(* LS Electric XG5000 project: Coffee_make *)
(* PLC LSPLC *)

(* Comments on direct variables
%MX1	원두리필시작
%MX2	원두부족알림
%MX3	물리필시작
%MX4	물부족알림
%MX5	우유리필시작
%MX6	우유부족알림
%MX7	초코부족알림
%MX8	카페부족알림
%MX9	물부족팝업
%MX10	원두부족팝업
%MX11	우유부족팝업
%MX21	환기
*)

PROGRAM NewProgram (* task: 스캔 프로그램 *)
VAR
    on AT %IX0.0.0 : BOOL;
    timer : TON;
    timer10 : TON;
    timer11 : TON;
    timer12 : TON;
    timer13 : TON;
    timer14 : TON;
    timer17 : TP;
    timer17_1 : TON;
    timer18 : TP;
    timer18_1 : TON;
    timer19 : TP;
    timer19_1 : TON;
    timer2 : TON;
    timer3 : TON;
    timer4 : TON;
    timer5 : TON;
    timer6 : TON;
    timer7 : TON;
    timer8 : TON;
    timer9 : TON;
    tp : TP;
    tp1 : TP;
    tp2 : TP;
    tp3 : TP;
    tp4 : TP;
    가스경고 : BOOL;
    경찰신고 AT %MX81 : BOOL;
    공기정화 AT %MX22 : BOOL;
    근접센서1 AT %MX450 : BOOL;
    근접센서2 : BOOL;
    끊어줌 : BOOL;
    끊어줌_TOF : TOF;
    끓인물투입통과 : BOOL;
    나감 AT %IX0.0.24 : BOOL;
    다음으로 : BOOL;
    다음으로자가유지 : BOOL;
    대형1층동작 : TON;
    대형감지 AT %MX455 : BOOL;
    대형감지완료 AT %MX452 : BOOL;
    대형나감_TON : TON;
    대형도착 AT %QX0.1.27 : BOOL;
    대형엘리동작1 : TON;
    대형입장 AT %IX0.0.22 : BOOL;
    대형자동차나감 AT %QX0.1.45 : BOOL;
    대형자동차나감유지 : BOOL;
    대형자동차이동1 AT %QX0.1.43 : BOOL;
    대형자동차이동1_TON : TON;
    대형자동차이동2 AT %QX0.1.44 : BOOL;
    대형자동차이동2_TON : TON;
    대형키오스크_TON : TON;
    대형키오스크이동 AT %QX0.1.42 : BOOL;
    대형키오스크자기유지 : BOOL;
    도착 AT %QX0.1.31 : BOOL;
    뜨거운물투입TPQ AT %MX39 : BOOL;
    레일동작1 AT %QX0.1.47 : BOOL;
    레일동작1_TON : TON;
    레일동작2 AT %QX0.1.48 : BOOL;
    레일동작2_TON : TON;
    레일동작3 AT %QX0.1.49 : BOOL;
    레일동작3_TON : TON;
    레일동작4 AT %QX0.1.50 : BOOL;
    레일동작4_TON : TON;
    레일정지 AT %QX0.1.24 : BOOL;
    매장경고음 AT %MX80 : BOOL;
    멈춤 AT %IX0.0.26 : BOOL;
    물 AT %MW22 : INT;
    물끓이기 : TON;
    물끓이기TP : TP;
    물끓이기TPQ AT %MX38 : BOOL;
    물끓이기여부 AT %MX18 : BOOL;
    물무게 AT %MW11 : INT;
    물무게UDINT : UDINT;
    물무게곱하기 : INT;
    물투입 : TON;
    물투입1 : TON;
    물투입1TP : TP;
    물투입1TPQ AT %MX45 : BOOL;
    물투입TP : TP;
    물투입시간 : TIME;
    물투입여부 : BOOL;
    물투입통과 : BOOL;
    사이안화수소 : INT;
    섞기 : TON;
    섞기TP : TP;
    섞기TPQ AT %MX36 : BOOL;
    섞기통과 : BOOL;
    소형감지 AT %MX457 : BOOL;
    소형감지완료 AT %MX454 : BOOL;
    소형나감_TON : TON;
    소형도착 AT %QX0.1.25 : BOOL;
    소형입장 AT %IX0.0.20 : BOOL;
    소형자동차나감 AT %QX0.1.36 : BOOL;
    소형자동차나감유지 : BOOL;
    소형자동차이동1 AT %QX0.1.34 : BOOL;
    소형자동차이동2 AT %QX0.1.35 : BOOL;
    소형키오스크_TON : TON;
    소형키오스크이동 AT %QX0.1.33 : BOOL;
    소형키오스크자기유지 : BOOL;
    스프링쿨러 : BOOL;
    시럽무게곱하기 : INT;
    시럽용우유투입통과 : BOOL;
    시럽우유무게UDINT : UDINT;
    시럽우유투입 : TON;
    시럽우유투입TP : TP;
    시럽우유투입TPQ AT %MX37 : BOOL;
    시럽우유투입시간 : TIME;
    시작 : BOOL;
    실링기계 : TON;
    실링기계동작 : BOOL;
    실링레일 : TON;
    실링레일동작 AT %QX0.1.46 : BOOL;
    안끓인물투입통과 : BOOL;
    알림전송 AT %MX82 : BOOL;
    어딘가 : BOOL;
    얼음선투입 AT %MX16 : BOOL;
    얼음선투입TP : TP;
    얼음선투입TPQ AT %MX31 : BOOL;
    얼음선투입타이머 : TON;
    얼음선투입통과 : BOOL;
    얼음후투입 AT %MX17 : BOOL;
    얼음후투입TP : TP;
    얼음후투입TPQ AT %MX42 : BOOL;
    얼음후투입타이머 : TON;
    얼음후투입통과 : BOOL;
    에이드액무게 : INT := 0;
    에이드투입 : BOOL := 0;
    엘리1층도착 : BOOL;
    엘리내려감 AT %QX0.1.30 : BOOL;
    엘리베이터대기 : TON;
    엘리베이터동작 AT %QX0.1.28 : BOOL;
    엘리베이터중지 AT %QX0.1.29 : BOOL;
    연화수소 : INT;
    온도경고 : BOOL;
    온도센서 AT %MW83 : INT;
    우유 AT %MW24 : INT;
    우유뎁히기 : TON;
    우유뎁히기TP : TP;
    우유뎁히기TPQ AT %MX34 : BOOL;
    우유무게 AT %MW12 : INT := 0;
    우유무게UDINT : UDINT;
    우유무게곱하기 : INT;
    우유투입 : TON;
    우유투입1 : TON;
    우유투입2 : TON;
    우유투입2TP : TP;
    우유투입2TPQ AT %MX46 : BOOL;
    우유투입3 : TON;
    우유투입TP : TP;
    우유투입TPQ AT %MX35 : BOOL;
    우유투입시간 : TIME;
    우유투입시작 : BOOL;
    우유투입여부 : BOOL;
    우유투입통과 : BOOL;
    원두 AT %MW20 : INT;
    원두갈기 : TON;
    원두넣기 : TON;
    원두넣기시간 : TIME := T#5s;
    원두추출 : TON;
    유독가스해결 AT %MX52 : BOOL;
    유독경고 : BOOL;
    유독스위치 AT %MX55 : BOOL;
    유독안전 : BOOL;
    유독유지 : BOOL;
    유독주의 : BOOL;
    음료제조시작 AT %IX0.0.1 : BOOL;
    음료제조완료 AT %QX0.1.0 : BOOL;
    음료제조자가유지 : BOOL;
    이산화탄소 AT %MW84 : INT;
    이상감지 : BOOL;
    인체경고 : BOOL;
    일단멈춰 AT %QX0.1.51 : BOOL;
    일단멈춰2 : BOOL;
    일단멈춰3 : BOOL;
    일단멈춰4 : BOOL;
    일단멈춰5 : BOOL;
    일단멈춰6 : BOOL;
    일단멈춰7 : BOOL;
    일단멈춰8 : BOOL;
    일반우유투입통과 : BOOL;
    일산화탄소 : INT;
    자동차이동1_TON : TON;
    자동차이동2_TON : TON;
    자동차입장감지센서 AT %QX0.1.20 : BOOL;
    재고물 AT %MW23 : INT;
    재고우유 AT %MW25 : INT;
    재고원두 AT %MW21 : INT;
    재고초코 AT %MW26 : INT;
    재고카페 AT %MW27 : INT;
    전력 AT %MX20 : BOOL;
    전력스위치 AT %MX50 : BOOL;
    주차차단기개방 AT %QX0.1.21 : BOOL;
    주차차단기차단 AT %QX0.1.37 : BOOL;
    중형1층동작 : TON;
    중형감지 AT %MX456 : BOOL;
    중형감지완료 AT %MX453 : BOOL;
    중형나감_TON : TON;
    중형도착 AT %QX0.1.26 : BOOL;
    중형엘리동작1 : TON;
    중형입장 AT %IX0.0.21 : BOOL;
    중형자동차나감 AT %QX0.1.41 : BOOL;
    중형자동차나감유지 : BOOL;
    중형자동차이동1 AT %QX0.1.39 : BOOL;
    중형자동차이동1_TON : TON;
    중형자동차이동2 AT %QX0.1.40 : BOOL;
    중형자동차이동2_TON : TON;
    중형키오스크_TON : TON;
    중형키오스크이동 AT %QX0.1.38 : BOOL;
    중형키오스크자기유지 : BOOL;
    지나감감지 : TON;
    차량나감 AT %QX0.1.52 : BOOL;
    초기화 AT %IX0.0.25 : BOOL;
    초코시럽무게 AT %MW13 : INT;
    초코시럽무게UDINT : UDINT;
    초코시럽무게곱하기 : INT;
    초코시럽투입 : TON;
    초코시럽투입TP : TP;
    초코시럽투입TPQ AT %MX33 : BOOL;
    초코시럽투입시간 : TIME;
    초코시럽투입여부 : BOOL;
    초코시럽투입통과 : BOOL;
    카페시럽무게 AT %MW14 : INT := 0;
    카페시럽무게UDINT : UDINT;
    카페시럽무게곱하기 : INT;
    카페시럽투입 : TON;
    카페시럽투입1 : TON;
    카페시럽투입2 : TON;
    카페시럽투입TP : TP;
    카페시럽투입TPQ AT %MX32 : BOOL;
    카페시럽투입시간 : TIME;
    카페시럽투입여부 : BOOL;
    카페시럽투입통과 : BOOL;
    커피가레일로 : TON;
    커피가레일로2 : TON;
    커피가레일로2TP : TP;
    커피가레일로2TPQ AT %MX44 : BOOL;
    커피가레일로TP : TP;
    커피가레일로TPQ AT %MX43 : BOOL;
    커피끓이기시간 : TIME;
    커피무게 AT %MW10 : INT;
    커피무게UDINT : UDINT;
    커피무게곱하기 : INT;
    커피배달중 AT %QX0.1.32 : BOOL;
    커피온도 AT %MW15 : INT;
    커피온도UDINT : UDINT;
    커피온도곱하기 : INT;
    커피제작시작 AT %QX0.1.22 : BOOL;
    커피제작완료 AT %QX0.1.23 : BOOL;
    커피주문완료 AT %MX451 : BOOL;
    커피추출 : TON;
    커피추출TP : TP;
    커피추출TPQ AT %MX40 : BOOL;
    커피투입 : TON;
    커피투입TP : TP;
    커피투입TPQ AT %MX41 : BOOL;
    커피투입시간 : TIME;
    커피투입시작 : BOOL;
    커피투입통과 : BOOL;
    컵구멍인지 : TON;
    컵투입 : TON;
    컵투입TP : TP;
    컵투입TPQ AT %MX30 : BOOL;
    컵투입통과 AT %MX65 : BOOL;
    컵투하직후TP : TP;
    쿨러온 AT %MX53 : BOOL;
    타이머 : TON;
    타이머1 : TON;
    타이머2 : TON;
    타이머3 : TON;
    호퍼닫기 : BOOL;
    화재위험 : BOOL;
    화재진압 : BOOL;
    환기스위치 AT %MX51 : BOOL;
END_VAR
VAR
    _t1 : BOOL;
    _t2 : BOOL;
    _t3 : BOOL;
    _t4 : BOOL;
    _p5 : BOOL;
    _t6 : BOOL;
    _t7 : BOOL;
    _t8 : BOOL;
    _t9 : BOOL;
    _t10 : BOOL;
    _t11 : BOOL;
    _t12 : BOOL;
    _t13 : BOOL;
    _t14 : BOOL;
    _t15 : BOOL;
    _t16 : BOOL;
    _t17 : BOOL;
END_VAR

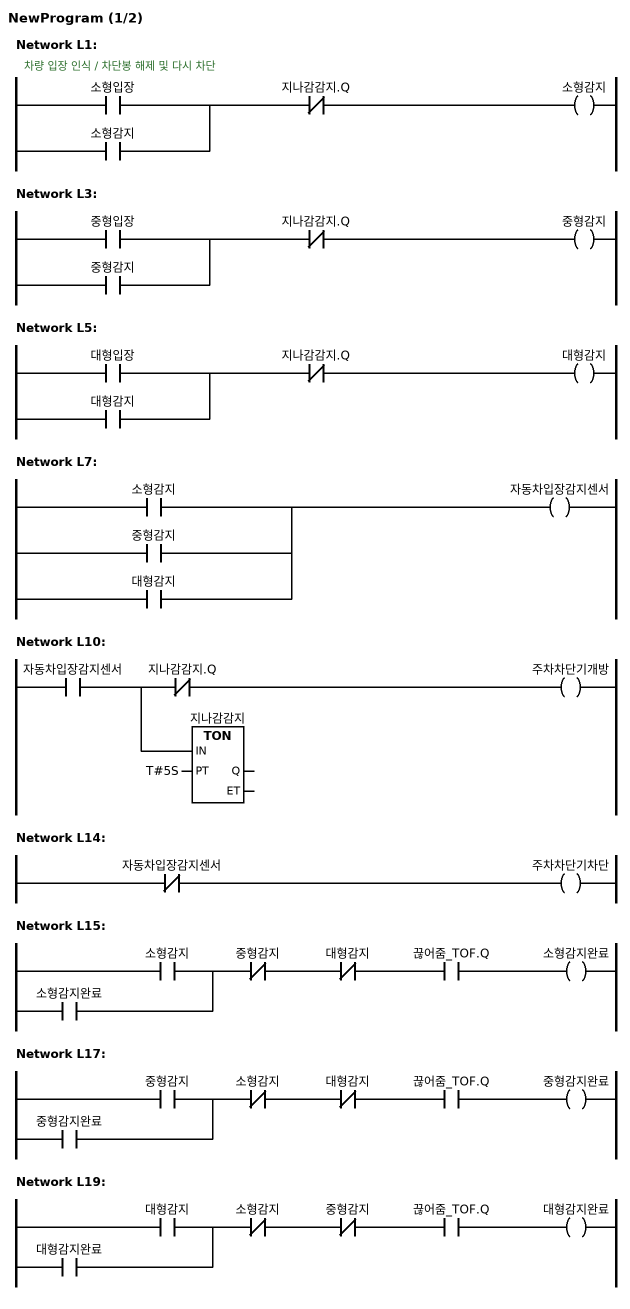
(* 차량 입장 인식 / 차단봉 해제 및 다시 차단 *)
(* Rung L1 *)
소형감지 := (소형입장 OR 소형감지) AND NOT 지나감감지.Q;
(* Rung L3 *)
중형감지 := (중형입장 OR 중형감지) AND NOT 지나감감지.Q;
(* Rung L5 *)
대형감지 := (대형입장 OR 대형감지) AND NOT 지나감감지.Q;
(* Rung L7 *)
자동차입장감지센서 := 소형감지 OR 중형감지 OR 대형감지;
(* Rung L10 *)
주차차단기개방 := 자동차입장감지센서 AND NOT 지나감감지.Q;
지나감감지(IN := 자동차입장감지센서, PT := T#5S);
(* Rung L14 *)
주차차단기차단 := NOT 자동차입장감지센서;
(* Rung L15 *)
소형감지완료 := (소형감지 OR 소형감지완료) AND NOT 중형감지 AND NOT 대형감지 AND 끊어줌_TOF.Q;
(* Rung L17 *)
중형감지완료 := (중형감지 OR 중형감지완료) AND NOT 소형감지 AND NOT 대형감지 AND 끊어줌_TOF.Q;
(* Rung L19 *)
대형감지완료 := (대형감지 OR 대형감지완료) AND NOT 소형감지 AND NOT 중형감지 AND 끊어줌_TOF.Q;

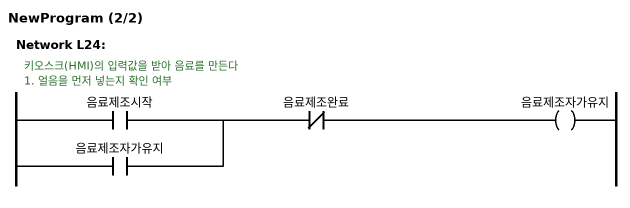
(* 키오스크(HMI)의 입력값을 받아 음료를 만든다 *)
(* 1. 얼음을 먼저 넣는지 확인 여부 *)
(* Rung L24 *)
음료제조자가유지 := (음료제조시작 OR 음료제조자가유지) AND NOT 음료제조완료;

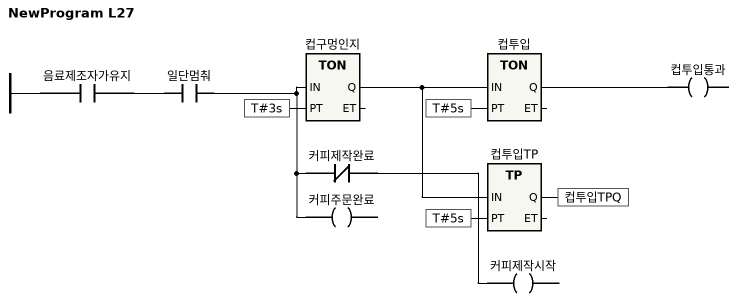
(* Rung L27 *)
커피제작시작 := 음료제조자가유지 AND 일단멈춰 AND NOT 커피제작완료;
커피주문완료 := 음료제조자가유지 AND 일단멈춰;
컵구멍인지(IN := 음료제조자가유지 AND 일단멈춰, PT := T#3s);
컵투입(IN := 컵구멍인지.Q, PT := T#5s);
컵투입통과 := 컵투입.Q;
컵투입TP(IN := 컵구멍인지.Q, PT := T#5s);
컵투입TPQ := 컵투입TP.Q;

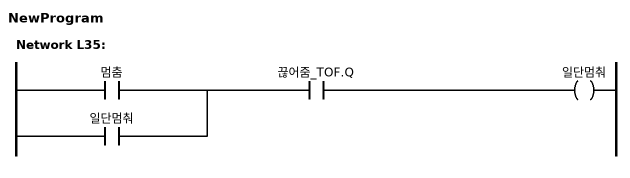
(* Rung L35 *)
일단멈춰 := (멈춤 OR 일단멈춰) AND 끊어줌_TOF.Q;

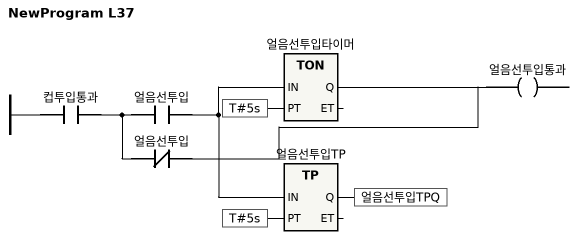
(* Rung L37 *)
얼음선투입타이머(IN := 컵투입통과 AND 얼음선투입, PT := T#5s);
얼음선투입통과 := 얼음선투입타이머.Q OR (컵투입통과 AND NOT 얼음선투입);
얼음선투입TP(IN := 컵투입통과 AND 얼음선투입, PT := T#5s);
얼음선투입TPQ := 얼음선투입TP.Q;

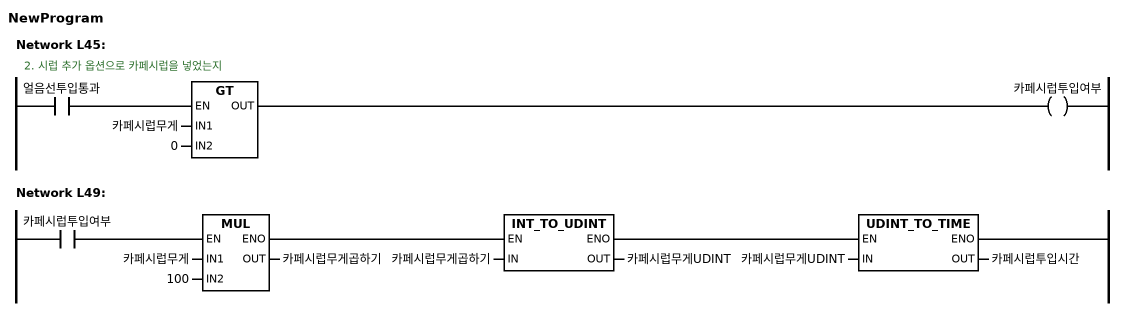
(* 2. 시럽 추가 옵션으로 카페시럽을 넣었는지 *)
(* Rung L45 *)
IF 얼음선투입통과 THEN _t1 := 카페시럽무게 > 0; END_IF;
카페시럽투입여부 := _t1;
(* Rung L49 *)
IF 카페시럽투입여부 THEN
    카페시럽무게곱하기 := 카페시럽무게 * 100;
    카페시럽무게UDINT := INT_TO_UDINT(카페시럽무게곱하기);
    카페시럽투입시간 := UDINT_TO_TIME(카페시럽무게UDINT);
END_IF;

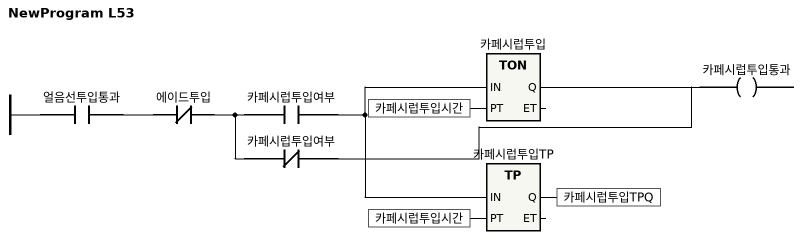
(* Rung L53 *)
카페시럽투입(IN := 얼음선투입통과 AND NOT 에이드투입 AND 카페시럽투입여부, PT := 카페시럽투입시간);
카페시럽투입통과 := 카페시럽투입.Q OR (얼음선투입통과 AND NOT 에이드투입 AND NOT 카페시럽투입여부);
카페시럽투입TP(IN := 얼음선투입통과 AND NOT 에이드투입 AND 카페시럽투입여부, PT := 카페시럽투입시간);
카페시럽투입TPQ := 카페시럽투입TP.Q;

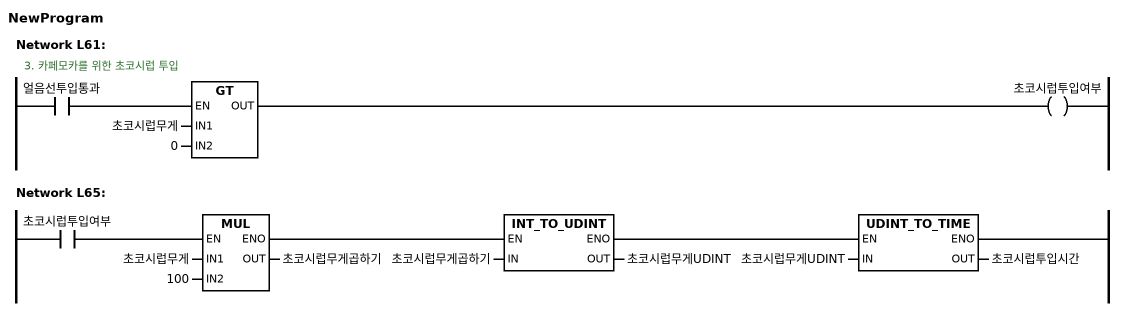
(* 3. 카페모카를 위한 초코시럽 투입 *)
(* Rung L61 *)
IF 얼음선투입통과 THEN _t2 := 초코시럽무게 > 0; END_IF;
초코시럽투입여부 := _t2;
(* Rung L65 *)
IF 초코시럽투입여부 THEN
    초코시럽무게곱하기 := 초코시럽무게 * 100;
    초코시럽무게UDINT := INT_TO_UDINT(초코시럽무게곱하기);
    초코시럽투입시간 := UDINT_TO_TIME(초코시럽무게UDINT);
END_IF;

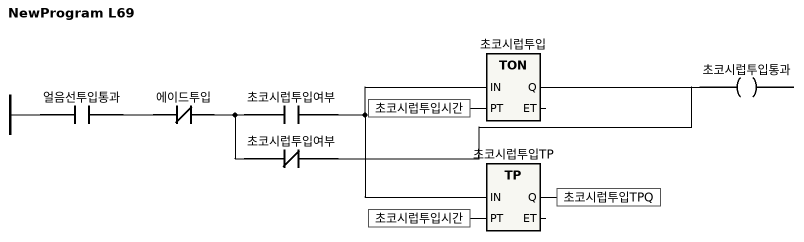
(* Rung L69 *)
초코시럽투입(IN := 얼음선투입통과 AND NOT 에이드투입 AND 초코시럽투입여부, PT := 초코시럽투입시간);
초코시럽투입통과 := 초코시럽투입.Q OR (얼음선투입통과 AND NOT 에이드투입 AND NOT 초코시럽투입여부);
초코시럽투입TP(IN := 얼음선투입통과 AND NOT 에이드투입 AND 초코시럽투입여부, PT := 초코시럽투입시간);
초코시럽투입TPQ := 초코시럽투입TP.Q;

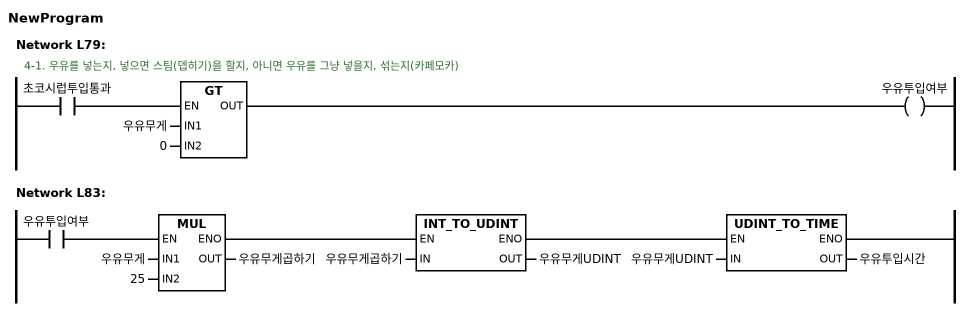
(* 4-1. 우유를 넣는지, 넣으면 스팀(뎁히기)을 할지, 아니면 우유를 그냥 넣을지, 섞는지(카페모카) *)
(* Rung L79 *)
IF 초코시럽투입통과 THEN _t3 := 우유무게 > 0; END_IF;
우유투입여부 := _t3;
(* Rung L83 *)
IF 우유투입여부 THEN
    우유무게곱하기 := 우유무게 * 25;
    우유무게UDINT := INT_TO_UDINT(우유무게곱하기);
    우유투입시간 := UDINT_TO_TIME(우유무게UDINT);
END_IF;

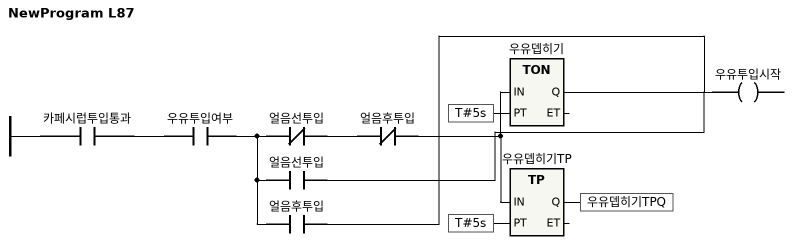
(* Rung L87 *)
우유뎁히기(IN := 카페시럽투입통과 AND 우유투입여부 AND NOT 얼음선투입 AND NOT 얼음후투입, PT := T#5s);
우유투입시작 := 우유뎁히기.Q OR (카페시럽투입통과 AND 우유투입여부 AND (얼음선투입 OR 얼음후투입));
우유뎁히기TP(IN := 카페시럽투입통과 AND 우유투입여부 AND NOT 얼음선투입 AND NOT 얼음후투입, PT := T#5s);
우유뎁히기TPQ := 우유뎁히기TP.Q;

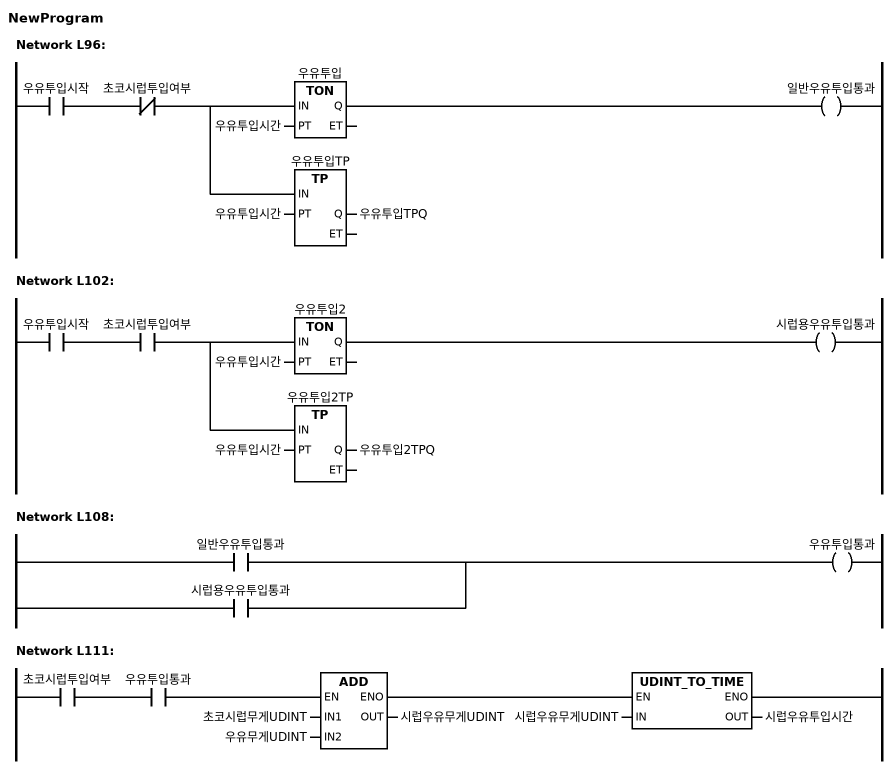
(* Rung L96 *)
우유투입(IN := 우유투입시작 AND NOT 초코시럽투입여부, PT := 우유투입시간);
일반우유투입통과 := 우유투입.Q;
우유투입TP(IN := 우유투입시작 AND NOT 초코시럽투입여부, PT := 우유투입시간, Q => 우유투입TPQ);
(* Rung L102 *)
우유투입2(IN := 우유투입시작 AND 초코시럽투입여부, PT := 우유투입시간);
시럽용우유투입통과 := 우유투입2.Q;
우유투입2TP(IN := 우유투입시작 AND 초코시럽투입여부, PT := 우유투입시간, Q => 우유투입2TPQ);
(* Rung L108 *)
우유투입통과 := 일반우유투입통과 OR 시럽용우유투입통과;
(* Rung L111 *)
IF 초코시럽투입여부 AND 우유투입통과 THEN
    시럽우유무게UDINT := 초코시럽무게UDINT + 우유무게UDINT;
    시럽우유투입시간 := UDINT_TO_TIME(시럽우유무게UDINT);
END_IF;

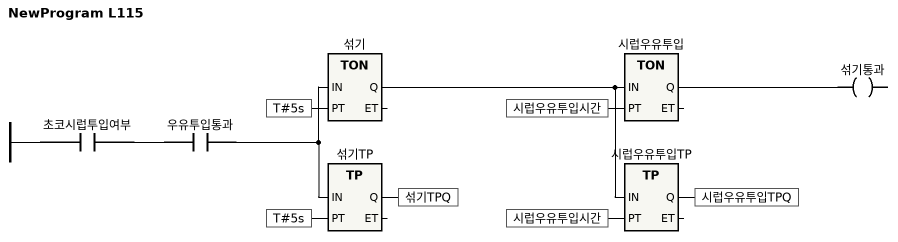
(* Rung L115 *)
섞기(IN := 초코시럽투입여부 AND 우유투입통과, PT := T#5s);
시럽우유투입(IN := 섞기.Q, PT := 시럽우유투입시간);
섞기통과 := 시럽우유투입.Q;
섞기TP(IN := 초코시럽투입여부 AND 우유투입통과, PT := T#5s);
섞기TPQ := 섞기TP.Q;
시럽우유투입TP(IN := 섞기.Q, PT := 시럽우유투입시간);
시럽우유투입TPQ := 시럽우유투입TP.Q;

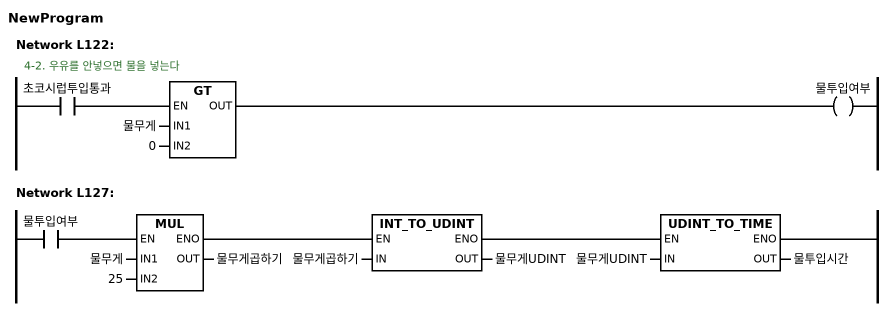
(* 4-2. 우유를 안넣으면 물을 넣는다 *)
(* Rung L122 *)
IF 초코시럽투입통과 THEN _t4 := 물무게 > 0; END_IF;
물투입여부 := _t4;
(* Rung L127 *)
IF 물투입여부 THEN
    물무게곱하기 := 물무게 * 25;
    물무게UDINT := INT_TO_UDINT(물무게곱하기);
    물투입시간 := UDINT_TO_TIME(물무게UDINT);
END_IF;

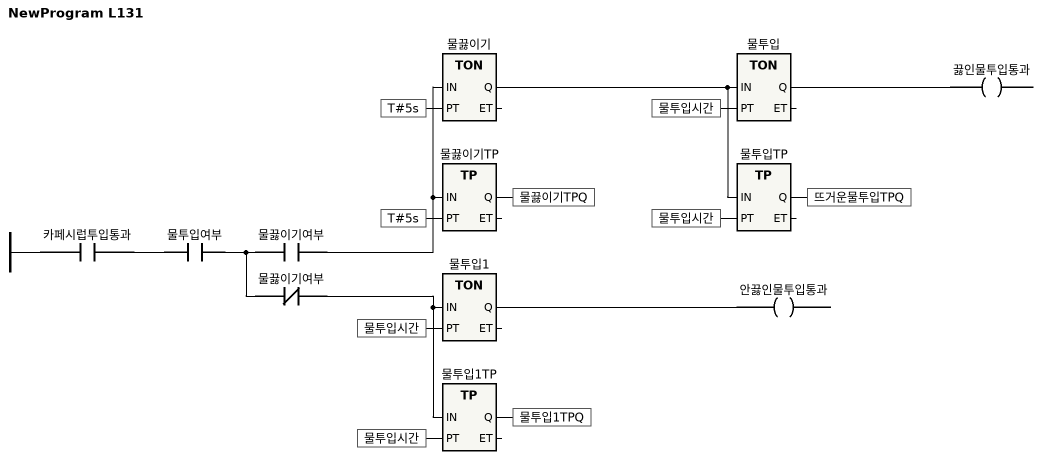
(* Rung L131 *)
물끓이기(IN := 카페시럽투입통과 AND 물투입여부 AND 물끓이기여부, PT := T#5s);
물투입(IN := 물끓이기.Q, PT := 물투입시간);
끓인물투입통과 := 물투입.Q;
물끓이기TP(IN := 카페시럽투입통과 AND 물투입여부 AND 물끓이기여부, PT := T#5s);
물끓이기TPQ := 물끓이기TP.Q;
물투입TP(IN := 물끓이기.Q, PT := 물투입시간);
뜨거운물투입TPQ := 물투입TP.Q;
물투입1(IN := 카페시럽투입통과 AND 물투입여부 AND NOT 물끓이기여부, PT := 물투입시간);
안끓인물투입통과 := 물투입1.Q;
물투입1TP(IN := 카페시럽투입통과 AND 물투입여부 AND NOT 물끓이기여부, PT := 물투입시간);
물투입1TPQ := 물투입1TP.Q;

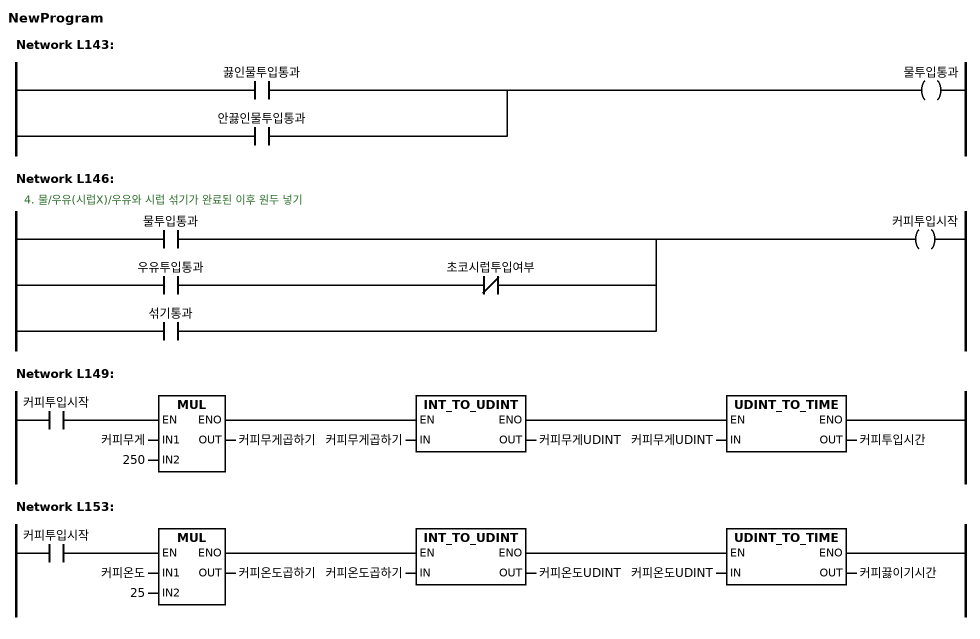
(* Rung L143 *)
물투입통과 := 끓인물투입통과 OR 안끓인물투입통과;
(* 4. 물/우유(시럽X)/우유와 시럽 섞기가 완료된 이후 원두 넣기 *)
(* Rung L146 *)
커피투입시작 := 물투입통과 OR (우유투입통과 AND NOT 초코시럽투입여부) OR 섞기통과;
(* Rung L149 *)
IF 커피투입시작 THEN
    커피무게곱하기 := 커피무게 * 250;
    커피무게UDINT := INT_TO_UDINT(커피무게곱하기);
    커피투입시간 := UDINT_TO_TIME(커피무게UDINT);
END_IF;
(* Rung L153 *)
IF 커피투입시작 THEN
    커피온도곱하기 := 커피온도 * 25;
    커피온도UDINT := INT_TO_UDINT(커피온도곱하기);
    커피끓이기시간 := UDINT_TO_TIME(커피온도UDINT);
END_IF;

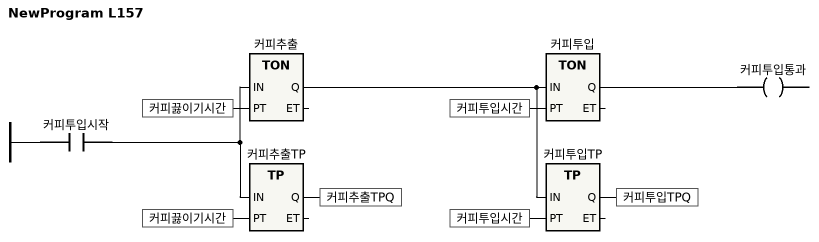
(* Rung L157 *)
커피추출(IN := 커피투입시작, PT := 커피끓이기시간);
커피투입(IN := 커피추출.Q, PT := 커피투입시간);
커피투입통과 := 커피투입.Q;
커피추출TP(IN := 커피투입시작, PT := 커피끓이기시간);
커피추출TPQ := 커피추출TP.Q;
커피투입TP(IN := 커피추출.Q, PT := 커피투입시간);
커피투입TPQ := 커피투입TP.Q;

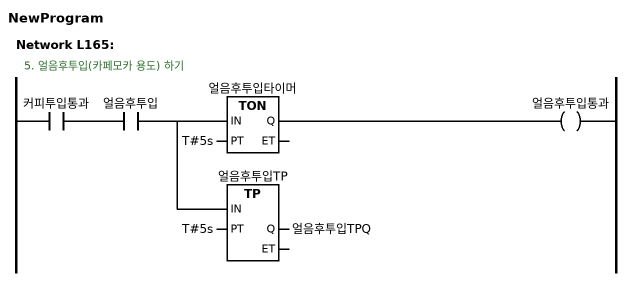
(* 5. 얼음후투입(카페모카 용도) 하기 *)
(* Rung L165 *)
얼음후투입타이머(IN := 커피투입통과 AND 얼음후투입, PT := T#5s);
얼음후투입통과 := 얼음후투입타이머.Q;
얼음후투입TP(IN := 커피투입통과 AND 얼음후투입, PT := T#5s, Q => 얼음후투입TPQ);

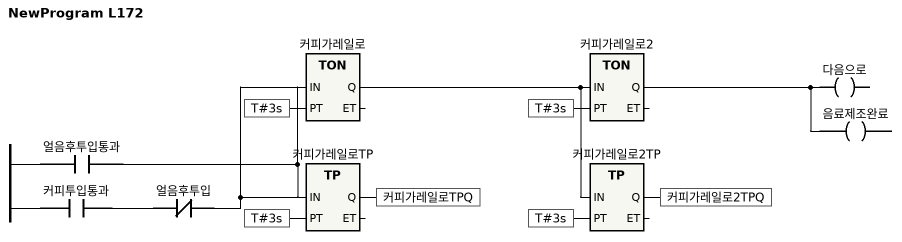
(* 끝. 음료제조완료 확인하기 *)
(* Rung L172 *)
커피가레일로(IN := 얼음후투입통과 OR (커피투입통과 AND NOT 얼음후투입), PT := T#3s);
커피가레일로2(IN := 커피가레일로.Q, PT := T#3s);
다음으로 := 커피가레일로2.Q;
음료제조완료 := 커피가레일로2.Q;
커피가레일로TP(IN := 얼음후투입통과 OR (커피투입통과 AND NOT 얼음후투입), PT := T#3s);
커피가레일로TPQ := 커피가레일로TP.Q;
커피가레일로2TP(IN := 커피가레일로.Q, PT := T#3s);
커피가레일로2TPQ := 커피가레일로2TP.Q;

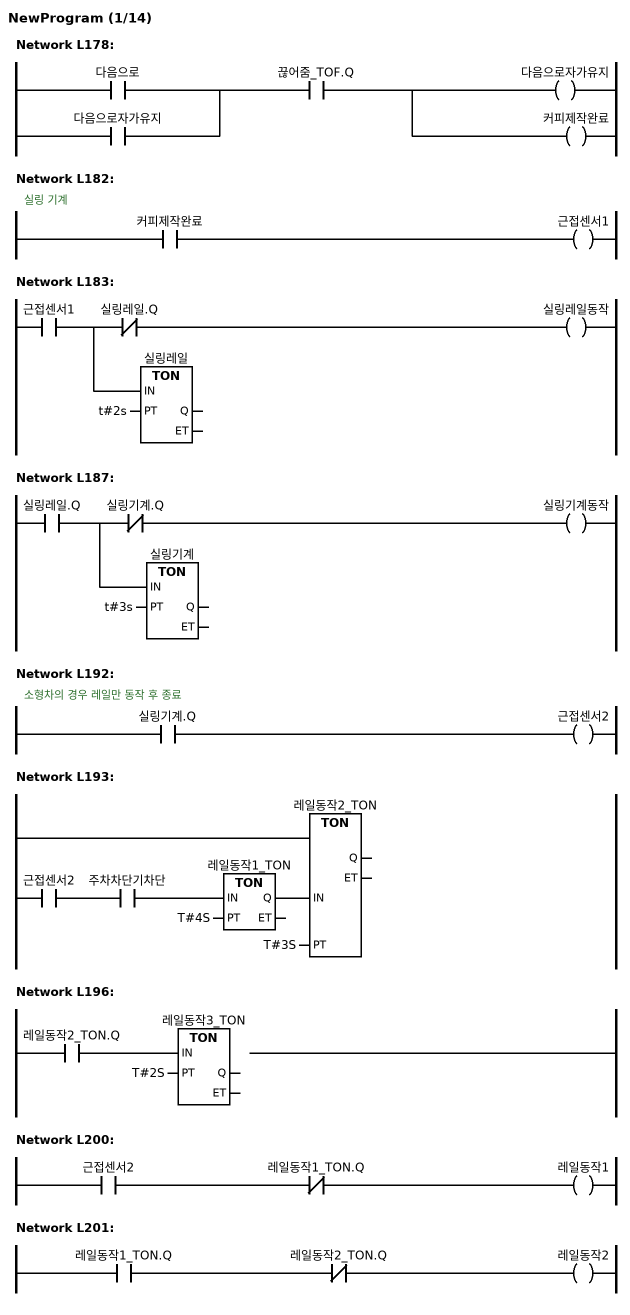
(* Rung L178 *)
_p5 := (다음으로 OR 다음으로자가유지) AND 끊어줌_TOF.Q;
다음으로자가유지 := _p5;
커피제작완료 := _p5;
(* 실링 기계 *)
(* Rung L182 *)
근접센서1 := 커피제작완료;
(* Rung L183 *)
실링레일동작 := 근접센서1 AND NOT 실링레일.Q;
실링레일(IN := 근접센서1, PT := t#2s);
(* Rung L187 *)
실링기계동작 := 실링레일.Q AND NOT 실링기계.Q;
실링기계(IN := 실링레일.Q, PT := t#3s);
(* 소형차의 경우 레일만 동작 후 종료 *)
(* Rung L192 *)
근접센서2 := 실링기계.Q;
(* Rung L193 *)
레일동작1_TON(IN := 근접센서2 AND 주차차단기차단, PT := T#4S);
레일동작2_TON(IN := 레일동작1_TON.Q, PT := T#3S);
(* Rung L196 *)
레일동작3_TON(IN := 레일동작2_TON.Q, PT := T#2S);
(* Rung L200 *)
레일동작1 := 근접센서2 AND NOT 레일동작1_TON.Q;
(* Rung L201 *)
레일동작2 := 레일동작1_TON.Q AND NOT 레일동작2_TON.Q;

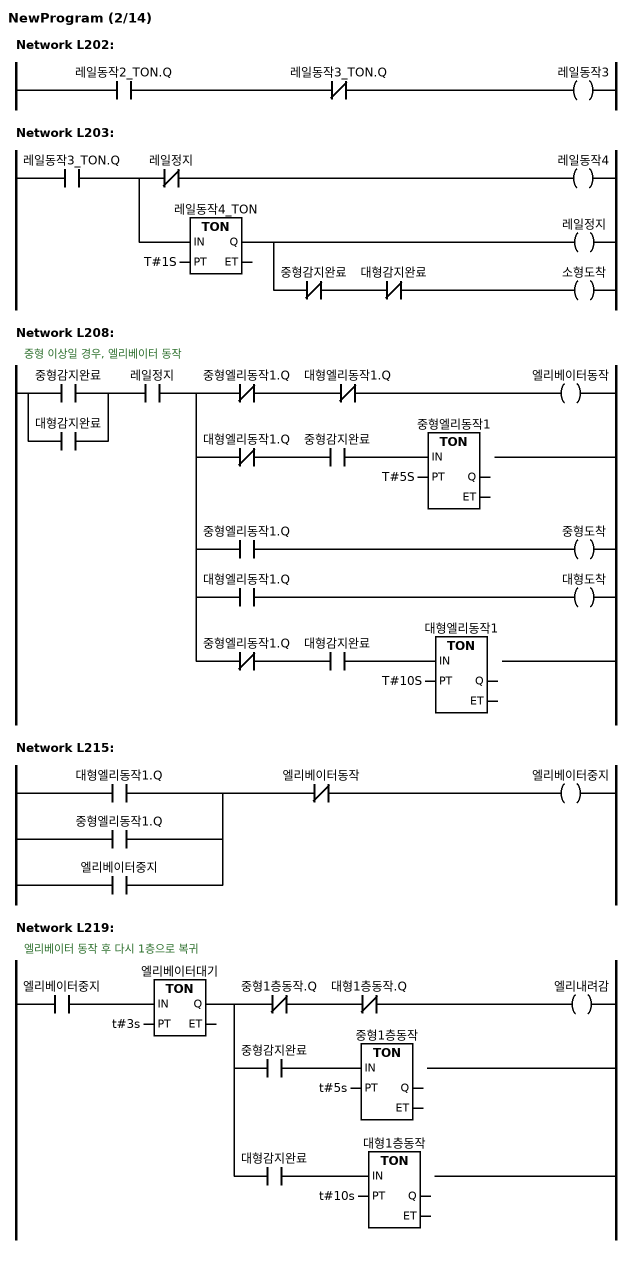
(* Rung L202 *)
레일동작3 := 레일동작2_TON.Q AND NOT 레일동작3_TON.Q;
(* Rung L203 *)
레일동작4 := 레일동작3_TON.Q AND NOT 레일정지;
레일동작4_TON(IN := 레일동작3_TON.Q, PT := T#1S);
레일정지 := 레일동작4_TON.Q;
소형도착 := 레일동작4_TON.Q AND NOT 중형감지완료 AND NOT 대형감지완료;
(* 중형 이상일 경우, 엘리베이터 동작 *)
(* Rung L208 *)
엘리베이터동작 := (중형감지완료 OR 대형감지완료) AND 레일정지 AND NOT 중형엘리동작1.Q AND NOT 대형엘리동작1.Q;
중형엘리동작1(IN := (중형감지완료 OR 대형감지완료) AND 레일정지 AND NOT 대형엘리동작1.Q AND 중형감지완료, PT := T#5S);
중형도착 := (중형감지완료 OR 대형감지완료) AND 레일정지 AND 중형엘리동작1.Q;
대형도착 := (중형감지완료 OR 대형감지완료) AND 레일정지 AND 대형엘리동작1.Q;
대형엘리동작1(IN := (중형감지완료 OR 대형감지완료) AND 레일정지 AND NOT 중형엘리동작1.Q AND 대형감지완료, PT := T#10S);
(* Rung L215 *)
엘리베이터중지 := (대형엘리동작1.Q OR 중형엘리동작1.Q OR 엘리베이터중지) AND NOT 엘리베이터동작;
(* 엘리베이터 동작 후 다시 1층으로 복귀 *)
(* Rung L219 *)
엘리베이터대기(IN := 엘리베이터중지, PT := t#3s);
엘리내려감 := 엘리베이터대기.Q AND NOT 중형1층동작.Q AND NOT 대형1층동작.Q;
중형1층동작(IN := 엘리베이터대기.Q AND 중형감지완료, PT := t#5s);
대형1층동작(IN := 엘리베이터대기.Q AND 대형감지완료, PT := t#10s);

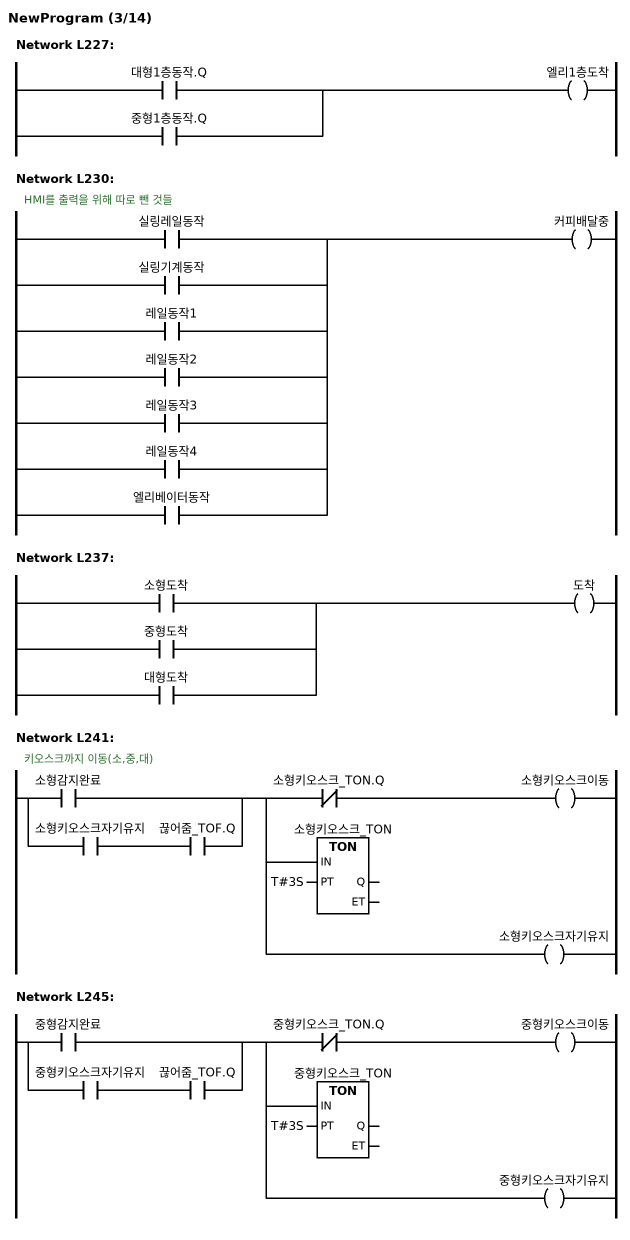
(* Rung L227 *)
엘리1층도착 := 대형1층동작.Q OR 중형1층동작.Q;
(* HMI를 출력을 위해 따로 뺀 것들 *)
(* Rung L230 *)
커피배달중 := 실링레일동작 OR 실링기계동작 OR 레일동작1 OR 레일동작2 OR 레일동작3 OR 레일동작4 OR 엘리베이터동작;
(* Rung L237 *)
도착 := 소형도착 OR 중형도착 OR 대형도착;
(* 키오스크까지 이동(소,중,대) *)
(* Rung L241 *)
소형키오스크이동 := (소형감지완료 OR (소형키오스크자기유지 AND 끊어줌_TOF.Q)) AND NOT 소형키오스크_TON.Q;
소형키오스크_TON(IN := 소형감지완료 OR (소형키오스크자기유지 AND 끊어줌_TOF.Q), PT := T#3S);
소형키오스크자기유지 := 소형감지완료 OR (소형키오스크자기유지 AND 끊어줌_TOF.Q);
(* Rung L245 *)
중형키오스크이동 := (중형감지완료 OR (중형키오스크자기유지 AND 끊어줌_TOF.Q)) AND NOT 중형키오스크_TON.Q;
중형키오스크_TON(IN := 중형감지완료 OR (중형키오스크자기유지 AND 끊어줌_TOF.Q), PT := T#3S);
중형키오스크자기유지 := 중형감지완료 OR (중형키오스크자기유지 AND 끊어줌_TOF.Q);

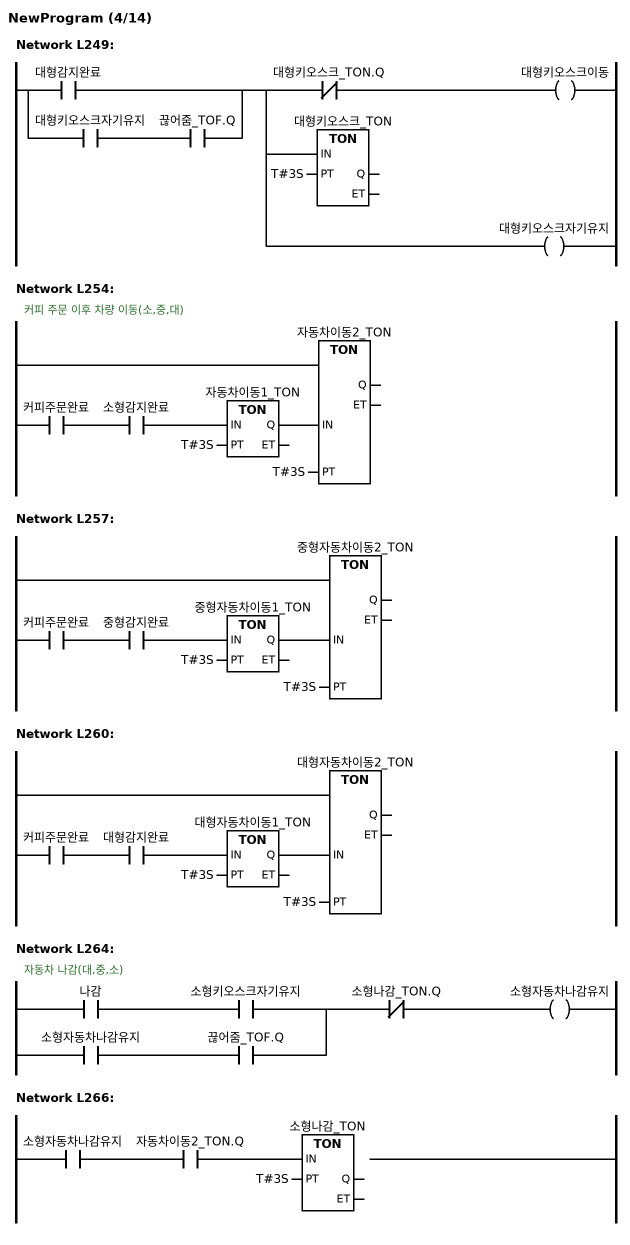
(* Rung L249 *)
대형키오스크이동 := (대형감지완료 OR (대형키오스크자기유지 AND 끊어줌_TOF.Q)) AND NOT 대형키오스크_TON.Q;
대형키오스크_TON(IN := 대형감지완료 OR (대형키오스크자기유지 AND 끊어줌_TOF.Q), PT := T#3S);
대형키오스크자기유지 := 대형감지완료 OR (대형키오스크자기유지 AND 끊어줌_TOF.Q);
(* 커피 주문 이후 차량 이동(소,중,대) *)
(* Rung L254 *)
자동차이동1_TON(IN := 커피주문완료 AND 소형감지완료, PT := T#3S);
자동차이동2_TON(IN := 자동차이동1_TON.Q, PT := T#3S);
(* Rung L257 *)
중형자동차이동1_TON(IN := 커피주문완료 AND 중형감지완료, PT := T#3S);
중형자동차이동2_TON(IN := 중형자동차이동1_TON.Q, PT := T#3S);
(* Rung L260 *)
대형자동차이동1_TON(IN := 커피주문완료 AND 대형감지완료, PT := T#3S);
대형자동차이동2_TON(IN := 대형자동차이동1_TON.Q, PT := T#3S);
(* 자동차 나감(대,중,소) *)
(* Rung L264 *)
소형자동차나감유지 := ((나감 AND 소형키오스크자기유지) OR (소형자동차나감유지 AND 끊어줌_TOF.Q)) AND NOT 소형나감_TON.Q;
(* Rung L266 *)
소형나감_TON(IN := 소형자동차나감유지 AND 자동차이동2_TON.Q, PT := T#3S);

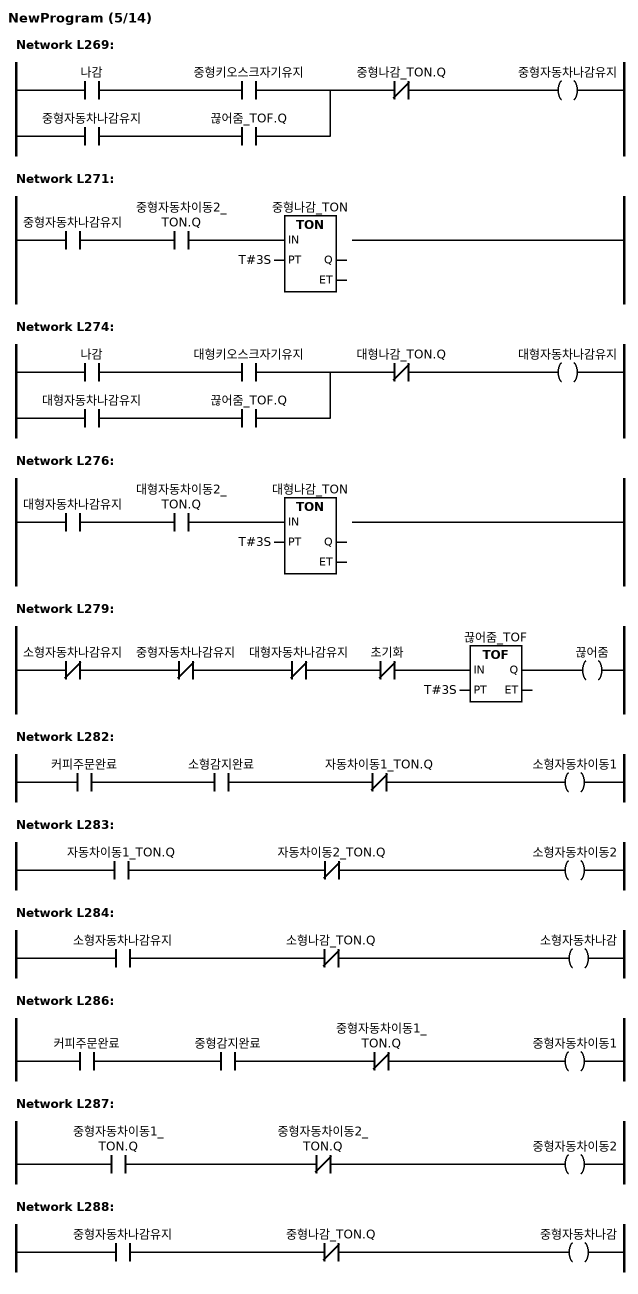
(* Rung L269 *)
중형자동차나감유지 := ((나감 AND 중형키오스크자기유지) OR (중형자동차나감유지 AND 끊어줌_TOF.Q)) AND NOT 중형나감_TON.Q;
(* Rung L271 *)
중형나감_TON(IN := 중형자동차나감유지 AND 중형자동차이동2_TON.Q, PT := T#3S);
(* Rung L274 *)
대형자동차나감유지 := ((나감 AND 대형키오스크자기유지) OR (대형자동차나감유지 AND 끊어줌_TOF.Q)) AND NOT 대형나감_TON.Q;
(* Rung L276 *)
대형나감_TON(IN := 대형자동차나감유지 AND 대형자동차이동2_TON.Q, PT := T#3S);
(* Rung L279 *)
끊어줌_TOF(IN := NOT 소형자동차나감유지 AND NOT 중형자동차나감유지 AND NOT 대형자동차나감유지 AND NOT 초기화, PT := T#3S);
끊어줌 := 끊어줌_TOF.Q;
(* Rung L282 *)
소형자동차이동1 := 커피주문완료 AND 소형감지완료 AND NOT 자동차이동1_TON.Q;
(* Rung L283 *)
소형자동차이동2 := 자동차이동1_TON.Q AND NOT 자동차이동2_TON.Q;
(* Rung L284 *)
소형자동차나감 := 소형자동차나감유지 AND NOT 소형나감_TON.Q;
(* Rung L286 *)
중형자동차이동1 := 커피주문완료 AND 중형감지완료 AND NOT 중형자동차이동1_TON.Q;
(* Rung L287 *)
중형자동차이동2 := 중형자동차이동1_TON.Q AND NOT 중형자동차이동2_TON.Q;
(* Rung L288 *)
중형자동차나감 := 중형자동차나감유지 AND NOT 중형나감_TON.Q;

